FUNCTION_BLOCK To_InfluxDb

VAR_INPUT
	bExecute: BOOL;		// Start logging when high. 
	tInterval: TIME;	// How often to log.
	sHostName: STRING;	// Ip-adress to Db
	nHostPort: UINT; // Influxdb is at 8086 default 
	sDatabaseName: STRING; // Db name
	sMeasurementName: STRING; // "Tablename"
	stData: ARRAY[0..10] OF ST_SensorData; // Data to be logged 
END_VAR
VAR_OUTPUT
	bBusy: BOOL;
	bError: BOOL;
	nErrId: DINT;
END_VAR
VAR
	nIndex: INT;
	nState: INT;
	nErrState: INT;
	sUri: STRING;
	sContent: STRING(32768);
	sData: STRING(255);
	nStartPos: UDINT;
	nLen: UDINT;
	
	tIntervalTimer: TON;
	fbIotHttpClient: FB_IotHttpClient;
	fbIotHttpRequest: FB_IotHttpRequest;
END_VAR

tIntervalTimer(IN:=bExecute AND NOT tIntervalTimer.Q, PT:=tInterval); // Timer for executing the http request.
CASE nState OF
0:	

	IF bExecute THEN
		bBusy:=TRUE;
		bError:=FALSE;
		nState:=10;
	END_IF

10:	

	mInit(); // Initialize HttpClient

20:

	mGenerateBodyContent(); // Generate data string to be sent to InfluxDb
	
21:

	mSendRequest(); // Execute send request
	
22:
	
	mWaitUntilDone(); // Wait until done or error

99:

	mErrorHandling(); // Handle the error if needed.
	
END_CASE

METHOD PRIVATE mErrorHandling : BOOL
bError:=TRUE;
bBusy:=FALSE;
IF NOT bExecute THEN
	nState:=0;
END_IF
END_METHOD

METHOD PRIVATE mGenerateBodyContent : BOOL
IF bExecute THEN
	IF tIntervalTimer.Q THEN
		sUri:=CONCAT('/write?db=', sDatabaseName);
		MEMSET(ADR(sContent),0,SIZEOF(sContent)); // Memset fixed the problems with status 400 and database havoc... 
		nStartPos:=0;
		FOR nIndex:=0 TO 5 DO
			IF stData[nIndex].sSensorId <> '' THEN
				sData:=sMeasurementName; 									nLen:=INT_TO_UDINT(LEN(sData)); MEMMOVE(ADR(sContent)+nStartPos, ADR(sData), nLen); nStartPos:=nStartPos+nLen;
				sData:=',SensorId='; 										nLen:=INT_TO_UDINT(LEN(sData)); MEMMOVE(ADR(sContent)+nStartPos, ADR(sData), nLen); nStartPos:=nStartPos+nLen;
				sData:=stData[nIndex].sSensorId; 							nLen:=INT_TO_UDINT(LEN(sData)); MEMMOVE(ADR(sContent)+nStartPos, ADR(sData), nLen); nStartPos:=nStartPos+nLen;
				sData:=' fSensorValue=';									nLen:=INT_TO_UDINT(LEN(sData)); MEMMOVE(ADR(sContent)+nStartPos, ADR(sData), nLen); nStartPos:=nStartPos+nLen;
				sData:=REAL_TO_STRING(stData[nIndex].rSensorValue);			nLen:=INT_TO_UDINT(LEN(sData)); MEMMOVE(ADR(sContent)+nStartPos, ADR(sData), nLen); nStartPos:=nStartPos+nLen;
				sData:='$n'; 												nLen:=INT_TO_UDINT(LEN(sData)); MEMMOVE(ADR(sContent)+nStartPos, ADR(sData), nLen); nStartPos:=nStartPos+nLen;
			ELSE
				EXIT;
			END_IF
		END_FOR
		nState:=21;
	END_IF	
ELSE
	bBusy:=FALSE;
	nState:=0;
END_IF
END_METHOD

METHOD PRIVATE mInit : BOOL
fbIotHttpClient.sHostName:=sHostName;
fbIotHttpClient.nHostPort:=nHostPort;
fbIotHttpClient.bKeepAlive:=TRUE;
fbIotHttpClient.tConnectionTimeout:=T#10S;
fbIotHttpClient.Execute();
IF fbIotHttpClient.bConfigured THEN
	nState:=20;
ELSIF fbIotHttpClient.bError THEN
	nErrState:=nState;
	nErrId:=fbIotHttpClient.hrErrorCode;
	nState:=99;
END_IF
END_METHOD

METHOD PRIVATE mSendRequest : BOOL

fbIotHttpClient.Execute();	
IF fbIotHttpRequest.SendRequest(
	sUri:=sUri,
	fbClient:=fbIotHttpClient, 
	eRequestType:=ETcIotHttpRequestType.HTTP_POST, 
	pContent:=ADR(sContent), 
	nContentSize:=LEN2(ADR(sContent)), 0)
THEN
	nState:=22;
END_IF
END_METHOD

METHOD PRIVATE mWaitUntilDone : BOOL

fbIotHttpClient.Execute();	
IF fbIotHttpRequest.bError THEN
	nErrState:=nState;
	nErrId:=fbIotHttpRequest.eErrorId;
	nState:=99;
ELSIF NOT fbIotHttpRequest.bBusy THEN
	nState:=20;
END_IF
END_METHOD

END_FUNCTION_BLOCK

(* stored: Version 1.1.0.1, ProductVersion 3.1.4024.9
   POU To_InfluxDb: Id {353446b1-c24f-4967-9083-9bc2fc8bcbeb}, SpecialFunc None
   Method mErrorHandling: Id {31dd8b71-e449-49c1-bfe2-6c14fd5a78e4}
   Method mGenerateBodyContent: Id {8f26b204-0b8b-4ac7-9d41-ae2ce7f25197}
   Method mInit: Id {92802100-23ff-47d3-8fb7-4fae70fc282d}
   Method mSendRequest: Id {e9679ef6-66e4-4272-b825-e8b826878320}
   Method mWaitUntilDone: Id {742ace05-a870-4b79-adc2-fb94ef0b85a0} *)
